FUNCTION_BLOCK ReflectUnwrap IMPLEMENTS I_Unwrapper
VAR
	_x : UDINT;
	_y : UDINT;
END_VAR

METHOD Sample : BOOL
VAR_INPUT
	ImageWidth	: UDINT;
	ImageHeight : UDINT;
	XOffset		: UDINT;
	YOffset		: UDINT;
END_VAR

VAR_INST
	factor : UDINT;
	even   : DINT;
END_VAR
even := TRUNC((XOffset) / (ImageWidth)) MOD 2;
IF even = 0 THEN
	_x := XOffset - (TRUNC(XOffset / ImageWidth) * ImageWidth);
ELSIF even = 1 THEN
	_x := ImageWidth - (XOffset - (TRUNC(XOffset / ImageWidth) * ImageWidth));
END_IF

_y	   := YOffset MOD (ImageHeight - 1);
Sample := TRUE;
END_METHOD

PROPERTY X : UDINT
GET
X := _x;
END_GET
END_PROPERTY

PROPERTY Y : UDINT
GET
Y := _y;
END_GET
END_PROPERTY

END_FUNCTION_BLOCK

(* stored: Version 1.1.0.1
   POU ReflectUnwrap: Id {a0c698c2-0b17-4426-b89a-abd08a8802fe}, SpecialFunc None
   Method Sample: Id {ac85f539-f222-4929-acbe-87181cca1d98}
   Property X: Id {ea1c1b89-8205-4df9-9b7d-6074fa2b32c2}
   Get Get: Id {c8fc38b6-5df7-4023-8a54-6944c353264a}
   Property Y: Id {d877612d-8c0d-4a9f-9190-ea1b80c3e8c2}
   Get Get: Id {349e4d7e-8e1f-43c6-938d-b02c1f7291b7} *)
